TYPE ST_DCEAP :
STRUCT
	//eapDBColumnPCWLeakage					AT %Q* :BOOL;
	//eapDBColumnPCWSupplyLeakage    		AT %Q* :BOOL;
	//eapDBColumnPCWReturnLeakage    		AT %Q* :BOOL;
END_STRUCT
END_TYPE

(* stored: Version 1.1.0.1, ProductVersion 3.1.4022.18
   DUT ST_DCEAP: Id {e263f8b5-995a-44ea-b04c-c6dfc03129bc} *)
